// TIA Portal V17 export
// export: Created 2025-01-08T13:55:36.5894056Z, ExportSetting WithDefaults, DisplayName Totally Integrated Automation Portal, DisplayVersion V17, DisplayName TIA Portal Openness, DisplayVersion V17, DisplayName TIA Portal Version Control Interface, DisplayVersion V17, DisplayName SINAMICS Startdrive Advanced, DisplayVersion V17 Update2, DisplayName SINAMICS Startdrive G130, G150, S120, S150, SINAMICS MV, S210, DisplayVersion V17 Update2, DisplayName SINAMICS Startdrive G110M, G120, G120C, G120D, G120P, G115D, DisplayVersion V17 Update2, DisplayName STEP 7 Professional, DisplayVersion V17, DisplayName STEP 7 Safety, DisplayVersion V17, DisplayName WinCC Advanced, DisplayVersion V17
TYPE "HSM_AlarmWarning"
// stored: IsFailsafeCompliant false
   STRUCT
      WWarning_08_Rewinder_Almost_Full : Bool;   // Rewinder almost full. Do a controlled stop and change otherwise machine may stop unexpected.
      WWarning_09_Roll_End_1 : Bool;
      WWarning_10_Roll_End_2 : Bool;
      WWarning_11_Roll_End_3 : Bool;
      WWarning_12 : Bool;
      WWarning_13 : Bool;
      WWarning_14 : Bool;
      WWarning_15 : Bool;
      WWarning_00 : Bool;
      WWarning_01_Find_Rotor_Position : Bool;   // Warning Rotor Position. Try restart.
      WWarning_02 : Bool;
      WWarning_03_Number_Of_Labels_Reached : Bool;   // This message indicates that the "Countdown" function has run to the end and has reached the end value "000".
      WWarning_04_Low_Label_Reached : Bool;   // This message indicates that the pre-set minimum diameter of the label roll for optional low label warning has been reached. When the residual label length (machine parameter [025] has been entered, the labeling mode is continued until this value has been reached. Thereafter, the labeler will stop and the "Web end reached” error message will be dis-played.
      WWarning_05_ZeroDownTime_Lan_Link_timeout : Bool;
      WWarning_06_ZeroDownTime_Parameter_error : Bool;
      WWarning_07 : Bool;
      AAlarm_14_Motor_Overcurrent : Bool;   // This message implies that the strain on the motor controller by the maximum current is too high. Potential causes: Too high cycle rate, paper brake to tight, material wrapped around the drive unit. Solution: Switch off the labeler, repair fault, switch on the labeler.
      AAlarm_15_Dancer_Arm_Stop_Reached : Bool;   // Unwinder dancer arm reached end position. End of label roll.
      AAlarm_16_Rewinder_Full : Bool;   // Rewinder full. Remove backing paper from rewinder and reattach to rewinder.
      AAlarm_17_Rewinder_Web_Break : Bool;   // Backing paper (web) broke or not attached to rewinder.
      AAlarm_18 : Bool;
      AAlarm_19 : Bool;
      AAlarm_20 : Bool;
      AAlarm_21 : Bool;
      AAlarm_6 : Bool;
      AAlarm_7_Motor_Start_Error : Bool;   // This message implies that the internal zero-compensation could not be performed. Switch off the labeler at the mains switch and wait until the display has gone off. Thereafter, switch the labeler back on.
      AAlarm_8_Motor_Position_Error : Bool;   // This message indicates that the servomotor cannot determine its rotor position during the initialization phase. Switch off the labeler at the mains switch and wait until the display has gone off. Thereafter, switch the labeler back on.
      AAlarm_9_Motor_Position_Control_Error : Bool;   // This message indicates that the servomotor cannot determine its prescribed position.
      AAlarm_10_Motor_Current_Target_Not_Reached : Bool;   // This message implies that the motor overload is too high, e.g. due to a short-circuit or ex-ternal interference.
      AAlarm_11_Label_Gap_Not_Found : Bool;   // This message implies that the label sensor does not detect the label stock. The existing labels between the label sensor and dispenser are dispensed completely. Thereafter, the system is switched to "Fault" (compare section above).
      AAlarm_12_Unwinder_Web_Break : Bool;   // This message means that the optional web break sensor detects that no label material is present. The currently applied label is still applied. Thereafter, the labeler interrupts the labeling cycle. Possible causes: Web break or end of web.
      AAlarm_13_Web_End : Bool;   // This message implies that the low label warning has been triggered and the pre-programmed residual label roll length (under machine parameter [025]) has lapsed. When the value for the remaining label length is set to "0" m (default value), a warning will be output but no "Error" triggered.
   END_STRUCT;
END_TYPE
